% RSLogix 500 project BELT_BAK000.RSS, saved by version 8.30.00.16 %
PROJECT "UNTITLED"    % processor: Bul.1763 MicroLogix 1100 Series B %

PROGRAM FILES
  LAD 2 "MAIN"  4 rungs
  LAD 3 "IO"  8 rungs
  LAD 4 "CTRL"  4 rungs
  LAD 5 "CYCLE"  10 rungs

DATA FILES
  O0 OUTPUT  4 elements
  I1 INPUT  6 elements
  S2 STATUS  66 elements
  B3 BINARY  2 elements
  T4 TIMER  1 elements
  C5 COUNTER  1 elements
  R6 CONTROL  1 elements
  N7 INTEGER  1 elements
  F8 FLOAT  1 elements

LADDER 2 "MAIN"
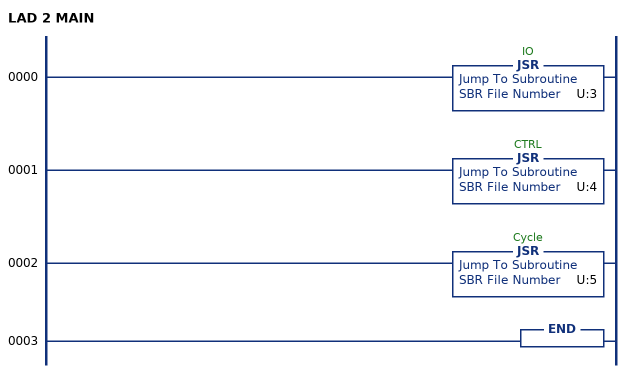
% Rung: 0 %
SOR JSR U:3 EOR
%   U:3  "IO" %
% Rung: 1 %
SOR JSR U:4 EOR
%   U:4  "CTRL" %
% Rung: 2 %
SOR JSR U:5 EOR
%   U:5  "Cycle" %
% Rung: 3 %
SOR END EOR

LADDER 3 "IO"
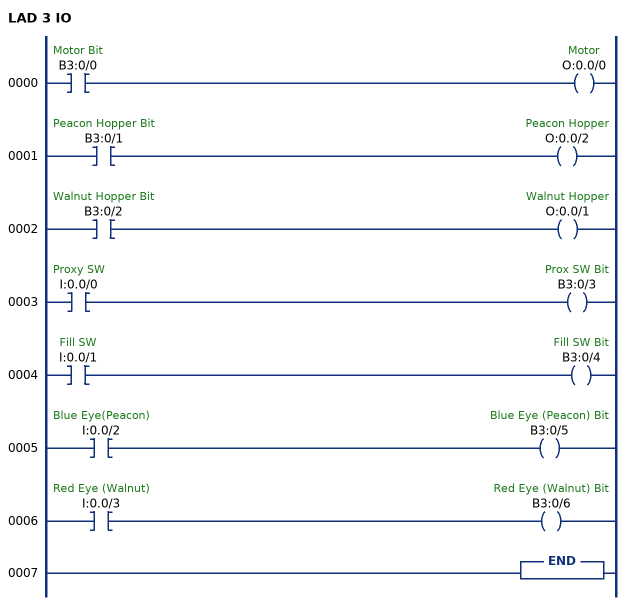
% Rung: 0 %
SOR XIC B3:0/0 OTE O:0.0/0 EOR
%   B3:0/0  "Motor Bit" %
%   O:0.0/0  "Motor" %
% Rung: 1 %
SOR XIC B3:0/1 OTE O:0.0/2 EOR
%   B3:0/1  "Peacon Hopper Bit" %
%   O:0.0/2  "Peacon Hopper" %
% Rung: 2 %
SOR XIC B3:0/2 OTE O:0.0/1 EOR
%   B3:0/2  "Walnut Hopper Bit" %
%   O:0.0/1  "Walnut Hopper" %
% Rung: 3 %
SOR XIC I:0.0/0 OTE B3:0/3 EOR
%   I:0.0/0  "Proxy SW" %
%   B3:0/3  "Prox SW Bit" %
% Rung: 4 %
SOR XIC I:0.0/1 OTE B3:0/4 EOR
%   I:0.0/1  "Fill SW" %
%   B3:0/4  "Fill SW Bit" %
% Rung: 5 %
SOR XIC I:0.0/2 OTE B3:0/5 EOR
%   I:0.0/2  "Blue Eye(Peacon)" %
%   B3:0/5  "Blue Eye (Peacon) Bit" %
% Rung: 6 %
SOR XIC I:0.0/3 OTE B3:0/6 EOR
%   I:0.0/3  "Red Eye (Walnut)" %
%   B3:0/6  "Red Eye (Walnut) Bit" %
% Rung: 7 %
SOR END EOR

LADDER 4 "CTRL"
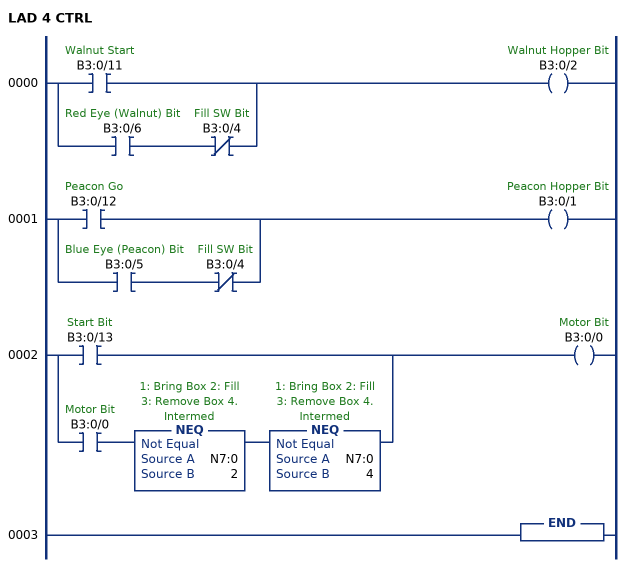
% Rung: 0 %
SOR BST XIC B3:0/11 NXB XIC B3:0/6 XIO B3:0/4 BND OTE B3:0/2 EOR
%   B3:0/11  "Walnut Start" %
%   B3:0/6  "Red Eye (Walnut) Bit" %
%   B3:0/4  "Fill SW Bit" %
%   B3:0/2  "Walnut Hopper Bit" %
% Rung: 1 %
SOR BST XIC B3:0/12 NXB XIC B3:0/5 XIO B3:0/4 BND OTE B3:0/1 EOR
%   B3:0/12  "Peacon Go" %
%   B3:0/5  "Blue Eye (Peacon) Bit" %
%   B3:0/4  "Fill SW Bit" %
%   B3:0/1  "Peacon Hopper Bit" %
% Rung: 2 %
SOR BST XIC B3:0/13 NXB XIC B3:0/0 NEQ N7:0 2 NEQ N7:0 4 BND OTE B3:0/0 EOR
%   B3:0/13  "Start Bit" %
%   B3:0/0  "Motor Bit" %
%   N7:0  "1: Bring Box 2: Fill 3: Remove Box 4. Intermed" %
% Rung: 3 %
SOR END EOR

LADDER 5 "CYCLE"
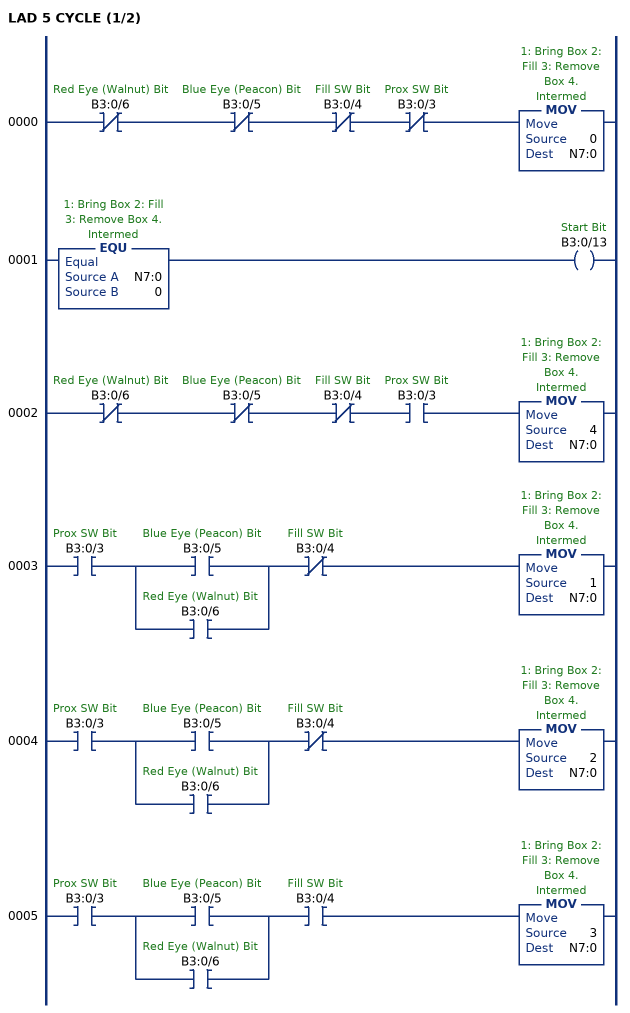
% Rung: 0 %
SOR XIO B3:0/6 XIO B3:0/5 XIO B3:0/4 XIO B3:0/3 MOV 0 N7:0 EOR
%   B3:0/6  "Red Eye (Walnut) Bit" %
%   B3:0/5  "Blue Eye (Peacon) Bit" %
%   B3:0/4  "Fill SW Bit" %
%   B3:0/3  "Prox SW Bit" %
%   N7:0  "1: Bring Box 2: Fill 3: Remove Box 4. Intermed" %
% Rung: 1 %
SOR EQU N7:0 0 OTE B3:0/13 EOR
%   N7:0  "1: Bring Box 2: Fill 3: Remove Box 4. Intermed" %
%   B3:0/13  "Start Bit" %
% Rung: 2 %
SOR XIO B3:0/6 XIO B3:0/5 XIO B3:0/4 XIC B3:0/3 MOV 4 N7:0 EOR
%   B3:0/6  "Red Eye (Walnut) Bit" %
%   B3:0/5  "Blue Eye (Peacon) Bit" %
%   B3:0/4  "Fill SW Bit" %
%   B3:0/3  "Prox SW Bit" %
%   N7:0  "1: Bring Box 2: Fill 3: Remove Box 4. Intermed" %
% Rung: 3 %
SOR XIC B3:0/3 BST XIC B3:0/5 NXB XIC B3:0/6 BND XIO B3:0/4 MOV 1 N7:0 EOR
%   B3:0/3  "Prox SW Bit" %
%   B3:0/5  "Blue Eye (Peacon) Bit" %
%   B3:0/6  "Red Eye (Walnut) Bit" %
%   B3:0/4  "Fill SW Bit" %
%   N7:0  "1: Bring Box 2: Fill 3: Remove Box 4. Intermed" %
% Rung: 4 %
SOR XIC B3:0/3 BST XIC B3:0/5 NXB XIC B3:0/6 BND XIO B3:0/4 MOV 2 N7:0 EOR
%   B3:0/3  "Prox SW Bit" %
%   B3:0/5  "Blue Eye (Peacon) Bit" %
%   B3:0/6  "Red Eye (Walnut) Bit" %
%   B3:0/4  "Fill SW Bit" %
%   N7:0  "1: Bring Box 2: Fill 3: Remove Box 4. Intermed" %
% Rung: 5 %
SOR XIC B3:0/3 BST XIC B3:0/5 NXB XIC B3:0/6 BND XIC B3:0/4 MOV 3 N7:0 EOR
%   B3:0/3  "Prox SW Bit" %
%   B3:0/5  "Blue Eye (Peacon) Bit" %
%   B3:0/6  "Red Eye (Walnut) Bit" %
%   B3:0/4  "Fill SW Bit" %
%   N7:0  "1: Bring Box 2: Fill 3: Remove Box 4. Intermed" %

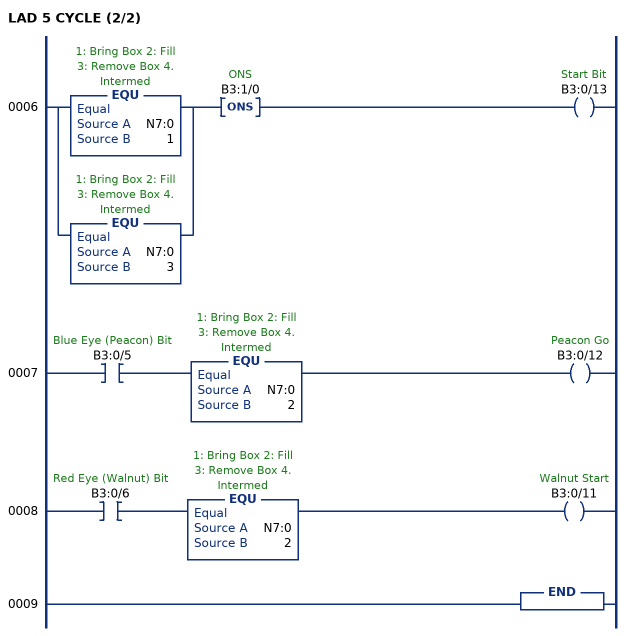
% Rung: 6 %
SOR BST EQU N7:0 1 NXB EQU N7:0 3 BND ONS B3:1/0 OTE B3:0/13 EOR
%   N7:0  "1: Bring Box 2: Fill 3: Remove Box 4. Intermed" %
%   B3:1/0  "ONS" %
%   B3:0/13  "Start Bit" %
% Rung: 7 %
SOR XIC B3:0/5 EQU N7:0 2 OTE B3:0/12 EOR
%   B3:0/5  "Blue Eye (Peacon) Bit" %
%   N7:0  "1: Bring Box 2: Fill 3: Remove Box 4. Intermed" %
%   B3:0/12  "Peacon Go" %
% Rung: 8 %
SOR XIC B3:0/6 EQU N7:0 2 OTE B3:0/11 EOR
%   B3:0/6  "Red Eye (Walnut) Bit" %
%   N7:0  "1: Bring Box 2: Fill 3: Remove Box 4. Intermed" %
%   B3:0/11  "Walnut Start" %
% Rung: 9 %
SOR END EOR

OTHER DOCUMENTED ADDRESSES
  B3:0/7  "Motor Go"
  B3:0/8  "Motor interupts"
  B3:0/9  "Fill stop"
  B3:0/15  "Motor start bit"
  B3:1/1  "ONS"
  B3:1/2  "ONS"
  T4:0  "Prox sw"
  T4:0/DN  "Prox SW Done"

DATA TABLE (non-zero values as saved)
DATA B3
% B3:0 % 0X00B8 0X0000
DATA T4
% .PRE .ACC %
% T4:0 % 0 50
DATA N7
% N7:0 % 3
